FUNCTION AnalayzeBatch : ST_ProductStats
VAR_INPUT
	aProdArray : REFERENCE TO ARRAY[1..20] OF REAL ;
END_VAR
VAR
	
END_VAR


AnalayzeBatch.fAverageWeight := CalculateAverage(aProdArray);
FindMinMax(aProdArray, fMinWeight => AnalayzeBatch.fminWeight, fMaxWeight => AnalayzeBatch.fmaxWeight);
AnalayzeBatch.nDefectiveCount := CountDefects(aProdArray);

END_FUNCTION

(* stored: Version 1.1.0.1, ProductVersion 3.1.4024.16
   POU AnalayzeBatch: Id {41693958-d985-4cab-8020-bde87749fe76}, SpecialFunc None *)
